INTERFACE I_ResponseIdGenerator

METHOD PUBLIC Generate : T_MAXSTRING
VAR_INPUT
END_VAR
END_METHOD

END_INTERFACE

(* stored: Version 1.1.0.1, ProductVersion 3.1.4024.12
   Itf I_ResponseIdGenerator: Id {dcb96cc9-2f85-4ac6-8d5e-482f2a92ec02}
   Method Generate: Id {c35c6504-c967-4797-9e3e-f6c5a8bfd9de} *)
